FUNCTION_BLOCK _ETcVnBarcodeSearchDirection_TestSuite EXTENDS TcUnit.FB_TestSuite
VAR
END_VAR

TestAddress();
TestClearReference();
TestClone();
TestTypeNameReturnsExpected();
TestIdentifierReturnsExpected();
TestMakeReferenceToFollowsReference();
TestMakeReferenceToUpdatesReference();
TestSize();
TestValueReturnsExpectedAfterInit();
TestValueReturnsExpectedAfterChange();
TestSerializeTypeWith();
TestSerializeWith();
TestTryDeserializeFrom();
TestTryMakeReferenceToFollowsReference();
TestTryMakeReferenceToUpdatesReference();

METHOD PUBLIC TestAddress
VAR
    _type : _ETcVnBarcodeSearchDirection(ETcVnBarcodeSearchDirection.TCVN_BSD_ANY);
    notExpected : PVOID := 0;
    actual : PVOID;
END_VAR
TEST('TestAddress');

actual := _type.Address;

AssertFalse(
    Condition := (notExpected = actual),
    Message := 'Type did not return a valid address.'
);

TEST_FINISHED();
END_METHOD

METHOD PUBLIC TestClearReference
VAR
    _type : _ETcVnBarcodeSearchDirection(ETcVnBarcodeSearchDirection.TCVN_BSD_ANY);
	target : ETcVnBarcodeSearchDirection := ETcVnBarcodeSearchDirection.TCVN_BSD_ANY;
    expected : ETcVnBarcodeSearchDirection := ETcVnBarcodeSearchDirection.TCVN_BSD_ANY;
    actual : ETcVnBarcodeSearchDirection;
END_VAR
TEST('TestClearReference');

_type.MakeReferenceTo(target);
_type.ClearReference();
target := ETcVnBarcodeSearchDirection.TCVN_BSD_HORIZONTAL;

actual := _type.Value;

AssertEquals(
    Expected := expected,
    Actual := actual,
    Message := 'Value continued to follow target.'
);

TEST_FINISHED();
END_METHOD

METHOD PUBLIC TestClone
VAR
    _type : _ETcVnBarcodeSearchDirection(ETcVnBarcodeSearchDirection.TCVN_BSD_ANY);
	clone : I_Datatype;
	isValidClone : BOOL;
	compareResult : DINT;
END_VAR
TEST('TestClone');

clone := _type.Clone();

isValidClone := clone <> 0;

IF isValidClone THEN
	compareResult := memcmp(_type.Address, clone.Address, clone.Size);
END_IF

AssertTrue(
	Condition := isValidClone,
	Message := 'Clone did not produce a clone'
);

AssertEquals_DINT(
	Expected := 0,
    Actual := compareResult,
    Message := 'Clone did not return a valid clone.'
);

clone.Dispose();

TEST_FINISHED();
END_METHOD

METHOD PUBLIC TestIdentifierReturnsExpected
VAR
    _type : _ETcVnBarcodeSearchDirection(ETcVnBarcodeSearchDirection.TCVN_BSD_ANY);
    expected : STRING := 'ETcVnBarcodeSearchDirection';
    actual : STRING;
END_VAR
TEST('TestIdentifierReturnsExpected');

actual := _type.Identifier;

AssertEquals_STRING(
    Expected := expected,
    Actual := actual,
    Message := 'Type did not return correct iec type.'
);

TEST_FINISHED();
END_METHOD

METHOD PUBLIC TestMakeReferenceToFollowsReference
VAR
    _type : _ETcVnBarcodeSearchDirection(ETcVnBarcodeSearchDirection.TCVN_BSD_ANY);
	target : ETcVnBarcodeSearchDirection := ETcVnBarcodeSearchDirection.TCVN_BSD_ANY;
    expected : ETcVnBarcodeSearchDirection := ETcVnBarcodeSearchDirection.TCVN_BSD_HORIZONTAL;
    actual : ETcVnBarcodeSearchDirection;
END_VAR
TEST('TestMakeReferenceToFollowsReference');

_type.MakeReferenceTo(target);
target := ETcVnBarcodeSearchDirection.TCVN_BSD_HORIZONTAL;

actual := _type.Value;

AssertEquals(
    Expected := expected,
    Actual := actual,
    Message := 'Value did not follow target change.'
);

TEST_FINISHED();
END_METHOD

METHOD PUBLIC TestMakeReferenceToUpdatesReference
VAR
    _type : _ETcVnBarcodeSearchDirection(ETcVnBarcodeSearchDirection.TCVN_BSD_ANY);
	target : ETcVnBarcodeSearchDirection := ETcVnBarcodeSearchDirection.TCVN_BSD_ANY;
    expected : ETcVnBarcodeSearchDirection := ETcVnBarcodeSearchDirection.TCVN_BSD_HORIZONTAL;
    actual : ETcVnBarcodeSearchDirection;
END_VAR
TEST('TestMakeReferenceToUpdatesReference');

_type.MakeReferenceTo(target);
_type.Value := ETcVnBarcodeSearchDirection.TCVN_BSD_HORIZONTAL;

actual := target;

AssertEquals(
    Expected := expected,
    Actual := actual,
    Message := 'Value did not update target.'
);

TEST_FINISHED();
END_METHOD

METHOD PUBLIC TestSerializeTypeWith
VAR
    _type : _ETcVnBarcodeSearchDirection(ETcVnBarcodeSearchDirection.TCVN_BSD_ANY);
    serializer : JsonSerializer;
    expected : STRING(500) := '{"typeName":"ENUM","identifier":"ETcVnBarcodeSearchDirection","enumerations":["TCVN_BSD_ANY","TCVN_BSD_HORIZONTAL","TCVN_BSD_VERTICAL"],"baseType":{"typeName":"UDINT","minValue":0,"maxValue":4294967295,"isSigned":false,"isFloat":false}}'; 
    actual : STRING(500);
END_VAR
TEST('TestSerializeTypeWith');

serializer.Reset();
_type.SerializeTypeWith(serializer);
serializer.TryGetSerializedData(ADR(actual), SIZEOF(actual));

AssertEquals_STRING(
    Expected := expected,
    Actual := actual,
    Message := 'Serialization of type did not return correct string.'
);

TEST_FINISHED();
END_METHOD

METHOD PUBLIC TestSerializeWith
VAR
    _type : _ETcVnBarcodeSearchDirection(ETcVnBarcodeSearchDirection.TCVN_BSD_ANY);
    serializer : JsonSerializer;
    expected : STRING := '"TCVN_BSD_ANY"';
    actual : STRING(500);
END_VAR
TEST('TestSerializeWith');

serializer.Reset();
_type.SerializeWith(serializer);
serializer.TryGetSerializedData(ADR(actual), SIZEOF(actual));

AssertEquals_STRING(
    Expected := expected,
    Actual := actual,
    Message := 'Serialization of type data did not return correct string.'
);

TEST_FINISHED();
END_METHOD

METHOD PUBLIC TestSize
VAR
    _type : _ETcVnBarcodeSearchDirection(ETcVnBarcodeSearchDirection.TCVN_BSD_ANY);
    expected : UDINT := SIZEOF(ETcVnBarcodeSearchDirection);
    actual : UDINT;
END_VAR
TEST('TestSize');

actual := _type.Size;

AssertEquals_UDINT(
    Expected := Expected,
    Actual := actual,
    Message := 'Type did not return the correct size.'
);

TEST_FINISHED();
END_METHOD

METHOD PUBLIC TestTryDeserializeFrom
VAR
    deserializer : JsonDeserializer;
    feedback : DeserializerFeedback;
    json : STRING := '"TCVN_BSD_ANY"';
    _type : _ETcVnBarcodeSearchDirection(ETcVnBarcodeSearchDirection.TCVN_BSD_ANY);
    expected : ETcVnBarcodeSearchDirection := ETcVnBarcodeSearchDirection.TCVN_BSD_ANY;
    actual : ETcVnBarcodeSearchDirection;
 END_VAR
TEST('TestTryDeserializeFrom');

deserializer.Reset();
deserializer.TryLoad(json);
_type.TryDeserializeFrom(Deserializer, Feedback);

actual := _type.Value;

AssertEquals(
    Expected := expected,
    Actual := actual,
    Message := 'Type did not deserialize correctly.'
);

TEST_FINISHED();
END_METHOD

METHOD PUBLIC TestTryMakeReferenceToFollowsReference
VAR
    _type : _ETcVnBarcodeSearchDirection(ETcVnBarcodeSearchDirection.TCVN_BSD_ANY);
	target : _ETcVnBarcodeSearchDirection(ETcVnBarcodeSearchDirection.TCVN_BSD_ANY);
    expected : ETcVnBarcodeSearchDirection := ETcVnBarcodeSearchDirection.TCVN_BSD_HORIZONTAL;
    actual : ETcVnBarcodeSearchDirection;
END_VAR
TEST('TestTryMakeReferenceToFollowsReference');

_type.TryMakeReferenceTo(target);
target.Value := ETcVnBarcodeSearchDirection.TCVN_BSD_HORIZONTAL;

actual := _type.Value;

AssertEquals(
    Expected := expected,
    Actual := actual,
    Message := 'Value did not follow target change.'
);

TEST_FINISHED();
END_METHOD

METHOD PUBLIC TestTryMakeReferenceToUpdatesReference
VAR
    _type : _ETcVnBarcodeSearchDirection(ETcVnBarcodeSearchDirection.TCVN_BSD_ANY);
	target : _ETcVnBarcodeSearchDirection(ETcVnBarcodeSearchDirection.TCVN_BSD_ANY);
    expected : ETcVnBarcodeSearchDirection := ETcVnBarcodeSearchDirection.TCVN_BSD_HORIZONTAL;
    actual : ETcVnBarcodeSearchDirection;
END_VAR
TEST('TestTryMakeReferenceToUpdatesReference');

_type.TryMakeReferenceTo(target);
_type.Value := ETcVnBarcodeSearchDirection.TCVN_BSD_HORIZONTAL;

actual := target.Value;

AssertEquals(
    Expected := expected,
    Actual := actual,
    Message := 'Value did not update target.'
);

TEST_FINISHED();
END_METHOD

METHOD PUBLIC TestTypeNameReturnsExpected
VAR
    _type : _ETcVnBarcodeSearchDirection(ETcVnBarcodeSearchDirection.TCVN_BSD_ANY);
    expected : STRING := 'ENUM';
    actual : STRING;
END_VAR
TEST('TestTypeNameReturnsExpected');

actual := _type.TypeName;

AssertEquals_STRING(
    Expected := expected,
    Actual := actual,
    Message := 'Type did not return correct iec type.'
);

TEST_FINISHED();
END_METHOD

METHOD PUBLIC TestValueReturnsExpectedAfterChange
VAR
    _type : _ETcVnBarcodeSearchDirection(ETcVnBarcodeSearchDirection.TCVN_BSD_ANY);
    expected : ETcVnBarcodeSearchDirection := ETcVnBarcodeSearchDirection.TCVN_BSD_HORIZONTAL;
    actual : ETcVnBarcodeSearchDirection;
END_VAR
TEST('TestValueReturnsExpectedAfterChange');

_type.Value := ETcVnBarcodeSearchDirection.TCVN_BSD_HORIZONTAL;

actual := _type.Value;

AssertEquals(
    Expected := expected,
    Actual := actual,
    Message := 'Expected value not returned after change.'
);

TEST_FINISHED();
END_METHOD

METHOD PUBLIC TestValueReturnsExpectedAfterInit
VAR
    _type : _ETcVnBarcodeSearchDirection(ETcVnBarcodeSearchDirection.TCVN_BSD_ANY);
    expected : ETcVnBarcodeSearchDirection := ETcVnBarcodeSearchDirection.TCVN_BSD_ANY;
    actual : ETcVnBarcodeSearchDirection;
END_VAR
TEST('TestValueReturnsExpectedAfterInit');

actual := _type.Value;

AssertEquals(
    Expected := expected,
    Actual := actual,
    Message := 'Expected value not returned after Init.'
);

TEST_FINISHED();
END_METHOD

END_FUNCTION_BLOCK

(* stored: Version 1.1.0.1, ProductVersion 3.1.4024.12
   POU _ETcVnBarcodeSearchDirection_TestSuite: Id {b842044a-e483-02e1-30ca-ae36851c9b06}, SpecialFunc None
   Method TestAddress: Id {717437e7-8721-0595-3e70-2a6b71643d53}
   Method TestClearReference: Id {00eeef00-914b-0807-0b0d-6d0d85c2aade}
   Method TestClone: Id {bd7390bf-c2cb-009b-20f4-d30364669dab}
   Method TestIdentifierReturnsExpected: Id {70825d47-8236-04c1-0d86-db1615962b4d}
   Method TestMakeReferenceToFollowsReference: Id {2da2bda5-0bc7-09ba-2b1e-624ef6e24240}
   Method TestMakeReferenceToUpdatesReference: Id {08879981-f5c6-06c2-1a0a-45294c6580d9}
   Method TestSerializeTypeWith: Id {ac771e29-6e18-0e09-26de-6556c1436722}
   Method TestSerializeWith: Id {aef96995-de79-0858-1887-b080e9e2f165}
   Method TestSize: Id {34e9c7f1-4dab-0e11-349f-73bac771e236}
   Method TestTryDeserializeFrom: Id {e9351961-d84e-0a89-1841-56c240540a01}
   Method TestTryMakeReferenceToFollowsReference: Id {91fb9d39-74af-03c8-370e-05ad3256a193}
   Method TestTryMakeReferenceToUpdatesReference: Id {a65cba03-082c-0684-16c0-325f4367d6e4}
   Method TestTypeNameReturnsExpected: Id {f2d13c96-27c4-002c-1a28-43b575dea5f2}
   Method TestValueReturnsExpectedAfterChange: Id {c2717a96-6b55-0931-0b1f-f3dc2e8e886c}
   Method TestValueReturnsExpectedAfterInit: Id {14c9fb6a-e391-00fd-31d5-26186c178494} *)
